FUNCTION_BLOCK JackHAL
  (* Standard: 61499-2 *)
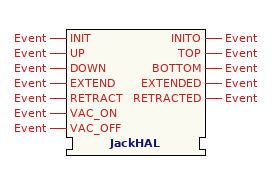
  EVENT_INPUT
    INIT;
    UP;
    DOWN;
    EXTEND;
    RETRACT;
    VAC_ON;
    VAC_OFF;
  END_EVENT
  EVENT_OUTPUT
    INITO;
    TOP;
    BOTTOM;
    EXTENDED;
    RETRACTED;
  END_EVENT
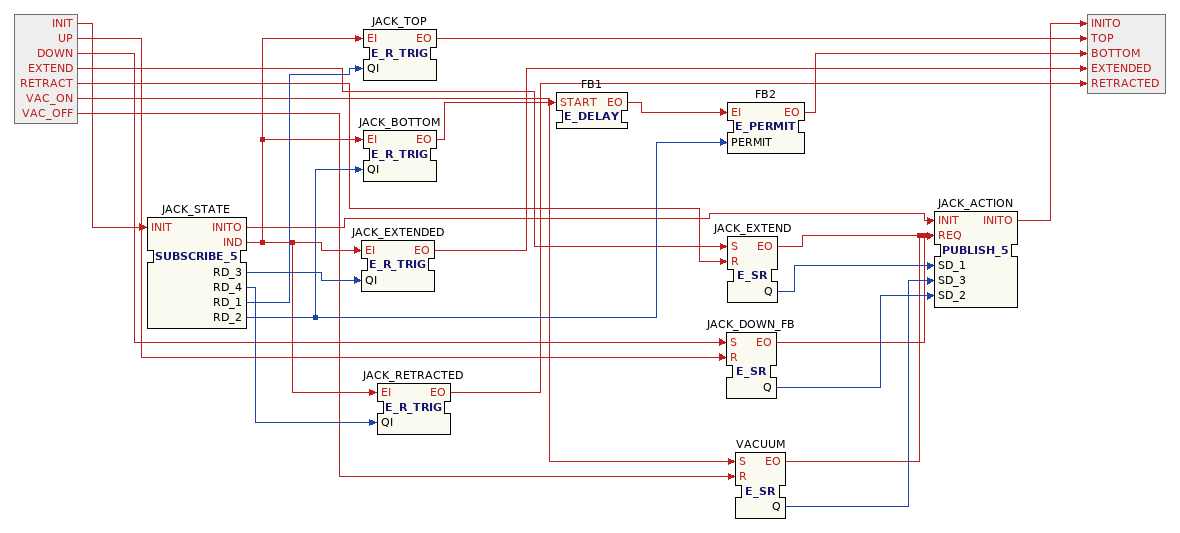
  FBS
    JACK_STATE : SUBSCRIBE_5;
    JACK_ACTION : PUBLISH_5;
    JACK_EXTEND : E_SR;
    JACK_DOWN_FB : E_SR;
    VACUUM : E_SR;
    JACK_EXTENDED : E_R_TRIG;
    JACK_RETRACTED : E_R_TRIG;
    JACK_TOP : E_R_TRIG;
    JACK_BOTTOM : E_R_TRIG;
    FB1 : E_DELAY;
    FB2 : E_PERMIT;
  END_FBS
  EVENT_CONNECTIONS
    INIT TO JACK_STATE.INIT;
    JACK_STATE.INITO TO JACK_ACTION.INIT;
    JACK_ACTION.INITO TO INITO;
    JACK_EXTEND.EO TO JACK_ACTION.REQ;
    EXTEND TO JACK_EXTEND.S;
    RETRACT TO JACK_EXTEND.R;
    DOWN TO JACK_DOWN_FB.S;
    UP TO JACK_DOWN_FB.R;
    JACK_DOWN_FB.EO TO JACK_ACTION.REQ;
    VACUUM.EO TO JACK_ACTION.REQ;
    VAC_ON TO VACUUM.S;
    VAC_OFF TO VACUUM.R;
    JACK_EXTENDED.EO TO EXTENDED;
    JACK_RETRACTED.EO TO RETRACTED;
    JACK_STATE.IND TO JACK_RETRACTED.EI;
    JACK_STATE.IND TO JACK_EXTENDED.EI;
    JACK_TOP.EO TO TOP;
    JACK_BOTTOM.EO TO FB1.START;
    JACK_STATE.IND TO JACK_TOP.EI;
    JACK_STATE.IND TO JACK_BOTTOM.EI;
    FB1.EO TO FB2.EI;
    FB2.EO TO BOTTOM;
  END_CONNECTIONS
  DATA_CONNECTIONS
    JACK_EXTEND.Q TO JACK_ACTION.SD_1;
    VACUUM.Q TO JACK_ACTION.SD_3;
    JACK_STATE.RD_3 TO JACK_EXTENDED.QI;
    JACK_STATE.RD_4 TO JACK_RETRACTED.QI;
    JACK_STATE.RD_1 TO JACK_TOP.QI;
    JACK_STATE.RD_2 TO JACK_BOTTOM.QI;
    JACK_STATE.RD_2 TO FB2.PERMIT;
    JACK_DOWN_FB.Q TO JACK_ACTION.SD_2;
  END_CONNECTIONS
END_FUNCTION_BLOCK
